(*

.. <legal notes>

legal notes
=================
| SPDX-FileCopyrightText: © 2026 Oleksandr Tiutyk <trofimich@gmail.com>
| SPDX-License-Identifier: LGPL-3.0-only
| For details check: LGPL-3.0-only_

.. _LGPL-3.0-only: https://www.gnu.org/licenses/lgpl-3.0.en.html

.. </legal notes>

*)

FUNCTION_BLOCK TrafficLight EXTENDS TOF_Automation.CompositeDevice<3> IMPLEMENTS TOF_Core.IIOBindable
VAR_OUTPUT
	RedLight : TOF_Devices_IO.DigitalOutput("RedLight", THIS^);
	YellowLight : TOF_Devices_IO.DigitalOutput("YellowLight", THIS^);
	GreenLight : TOF_Devices_IO.DigitalOutput("GreenLight", THIS^);
END_VAR
VAR
	_ClassName : STRING := __POUNAME();
	
	_SubDevices : ARRAY [0.._SubDeviceCount - 1] OF TOF_Automation.IDevice := 
	[
		RedLight, 
		YellowLight, 
		GreenLight
	];
END_VAR

METHOD BindToIO
VAR_INPUT
	redLightRawValue : REFERENCE TO BOOL;
	yellowLightRawValue : REFERENCE TO BOOL;
	greenLightRawValue : REFERENCE TO BOOL;
END_VAR
RedLight.BindToIO(redLightRawValue);
YellowLight.BindToIO(yellowLightRawValue);
GreenLight.BindToIO(greenLightRawValue);
END_METHOD

{attribute 'monitoring' := 'call'}
PROPERTY FINAL BoundToIO : BOOL
GET
BoundToIO := RedLight.BoundToIO AND_THEN YellowLight.BoundToIO AND_THEN GreenLight.BoundToIO;
END_GET
END_PROPERTY

{attribute 'monitoring' := 'call'}
PROPERTY ClassName : STRING
GET
ClassName := _ClassName;
END_GET
END_PROPERTY

{attribute 'monitoring' := 'call'}
PROPERTY NamespaceName : STRING
GET
NamespaceName := CurrentNamespace.Name;
END_GET
END_PROPERTY

{attribute 'monitoring' := 'call'}
PROPERTY SelfSize : ULINT
GET
SelfSize := XSIZEOF(THIS^);
END_GET
END_PROPERTY

METHOD SetLight
VAR_INPUT
	color : TRAFFIC_LIGHT_COLOR;
END_VAR
RedLight.Value := color = TRAFFIC_LIGHT_COLOR.RED;
YellowLight.Value := color = TRAFFIC_LIGHT_COLOR.YELLOW;
GreenLight.Value := color = TRAFFIC_LIGHT_COLOR.GREEN;
END_METHOD

PROPERTY SubDevices : REFERENCE TO ARRAY [0.._SubDeviceCount - 1] OF TOF_Automation.IDevice
GET
SubDevices REF= _SubDevices;
END_GET
END_PROPERTY

END_FUNCTION_BLOCK

(* stored: Version 1.1.0.1
   POU TrafficLight: Id {4a48deea-1b31-43e8-87e2-aa154a1466e2}, SpecialFunc None
   Method BindToIO: Id {55cb475d-9082-491a-a7db-c010249b1dee}
   Property BoundToIO: Id {59765228-75e5-4a28-a5ce-f29eb52a2c07}
   Get Get: Id {2a0ad00d-a286-4691-80b4-d1cec1c85bff}
   Property ClassName: Id {57d4725e-1474-4661-8746-ce344608dbc4}
   Get Get: Id {bf033ab4-a042-404c-85bc-755e1b6f3d73}
   Property NamespaceName: Id {4ef76813-685e-4906-ba01-6114c2c08566}
   Get Get: Id {03ffe5c5-1446-4400-87f1-63e337477d04}
   Property SelfSize: Id {0854c0b6-08bb-4062-b879-abc7c2048c2f}
   Get Get: Id {be673c01-8bac-444a-bd16-fa3be540c5df}
   Method SetLight: Id {66ac2472-cd7a-4221-b0c7-b8380631be67}
   Property SubDevices: Id {24d9159e-d58e-4242-9c68-13fddc2a3388}
   Get Get: Id {a8e5d14a-9275-4393-b35e-1978fe96fc18} *)
